(*

short summary
=================
This interface provides assert statements for times
For ``LTIME`` assertions use the property :ref:`ITimeAssertions.long`.
For ``TIME`` assertions use the property :ref:`ITimeAssertions.simple`.
.. <legal notes>

legal notes
=================
| SPDX-FileCopyrightText: © 2022 ekvip automation GmbH <info@ekvip.de>
| SPDX-License-Identifier: Apache-2.0
| For details check: Apache-2.0_

.. _Apache-2.0: https://www.apache.org/licenses/LICENSE-2.0

.. </legal notes>

methods
==================

*)

INTERFACE ITimeAssertions EXTENDS __SYSTEM.IQueryInterface

(*

short summary
=================
Returns an interface with assert statements for 64 bit times 

.. <legal notes>

legal notes
=================
| SPDX-FileCopyrightText: © 2022 ekvip automation GmbH <info@ekvip.de>
| SPDX-License-Identifier: Apache-2.0
| For details check: Apache-2.0_

.. _Apache-2.0: https://www.apache.org/licenses/LICENSE-2.0

.. </legal notes>

*)

PROPERTY long :I64BitTimeAssertions
GET
END_GET
END_PROPERTY

(*

short summary
=================
Returns an interface with assert statements for 32 bit times 

.. <legal notes>

legal notes
=================
| SPDX-FileCopyrightText: © 2022 ekvip automation GmbH <info@ekvip.de>
| SPDX-License-Identifier: Apache-2.0
| For details check: Apache-2.0_

.. _Apache-2.0: https://www.apache.org/licenses/LICENSE-2.0

.. </legal notes>

*)

PROPERTY simple :I32BitTimeAssertions
GET
END_GET
END_PROPERTY

END_INTERFACE

(* stored: Version 1.1.0.1, ProductVersion 3.1.4024.11
   Itf ITimeAssertions: Id {8deb3fdf-8e80-4673-b402-5f6d488ddd4a}
   Property long: Id {74e15394-1d52-45c6-bf5c-6f8ec91c4912}
   Get Get: Id {be0e63be-a117-431c-bbdd-3aa14aa6372b}
   Property simple: Id {c801510a-1f96-4735-a4d2-5ba37f80050c}
   Get Get: Id {5b374208-8957-45cf-bc27-2936a2069145} *)
